{attribute 'qualified_only'}
VAR_GLOBAL
	{attribute 'OPC.UA.DA' := '1'}	
	stFcuControl	: ST_FcuControl;
	
	{attribute 'OPC.UA.DA' := '1'}
	stSpindleControl	: ST_SpindleControl;
	
	{attribute 'OPC.UA.DA' := '1'}	
	stTestBasic	: ST_TestBasicControl;
END_VAR

(* stored: Version 1.1.0.1, ProductVersion 3.1.4024.9
   GVL GVL_opcua: Id {273b9490-171c-4ca8-b282-10eab17b1921} *)
